// TIA Portal V19 export
FUNCTION_BLOCK "DrvSafeSinaSTlg30"   // FB5, F_LAD
TITLE = SINAMICS S Safety Integrated Functions
// The library includes fail-safe S7 blocks to implement various applications in conjunction with S7-1200F, S7-1500F, S7-1500F Software Controller, SINUMERIK ONE and SINAMICS or SIMATIC Micro Drive coupled via PROFIsafe.
// Additional information in the application example "SIMATIC - Failsafe library LDrvSafe to control the Safety Integrated functions of the SINAMICS drive family"
// stored: IsIECCheckEnabled true, Namespace Safety
   VAR_INPUT
      ack { ExternalAccessible := 'False'; ExternalVisible := 'False'; ExternalWritable := 'False'} : Bool := false;   // Acknowledge bit
      sto { ExternalAccessible := 'False'; ExternalVisible := 'False'; ExternalWritable := 'False'} : Bool := true;   // 1: Deselect STO 0: Select STO
      ss1 { ExternalAccessible := 'False'; ExternalVisible := 'False'; ExternalWritable := 'False'} : Bool := true;   // 1: Deselect SS1 0: Select SS1
      sls { ExternalAccessible := 'False'; ExternalVisible := 'False'; ExternalWritable := 'False'} : Bool := true;   // 1: Deselect SLS 0: Select SLS
      statusWord { ExternalAccessible := 'False'; ExternalVisible := 'False'; ExternalWritable := 'False'} : "Safety.LDrvSafe_typeSinaSTlg30Status";   // PROFIsafe status telegram of the drive
   END_VAR
   VAR_OUTPUT
      status { ExternalAccessible := 'False'; ExternalVisible := 'False'; ExternalWritable := 'False'} : "Safety.typeSafetyDrive";
      controlWord { ExternalAccessible := 'False'; ExternalVisible := 'False'; ExternalWritable := 'False'} : "Safety.LDrvSafe_typeSinaSTlg30Control";   // PROFIsafe control telegram of the drive
   END_VAR
   VAR
      instLDrvSafeSinaSTlg30Status { ExternalAccessible := 'False'; ExternalVisible := 'False'; ExternalWritable := 'False'} : "Safety.LDrvSafe_SinaSTlg30Status";   // Instance data for status telegram
      instLDrvSafeSinaSTlg30Control { ExternalAccessible := 'False'; ExternalVisible := 'False'; ExternalWritable := 'False'} : "Safety.LDrvSafe_SinaSTlg30Control";   // Instance data for control telegram
   END_VAR
BEGIN

REGION Network 1: Control telegram
   // This block controls the safety integrated functions of a SINAMICS S drive via PROFIsafe telegram 30
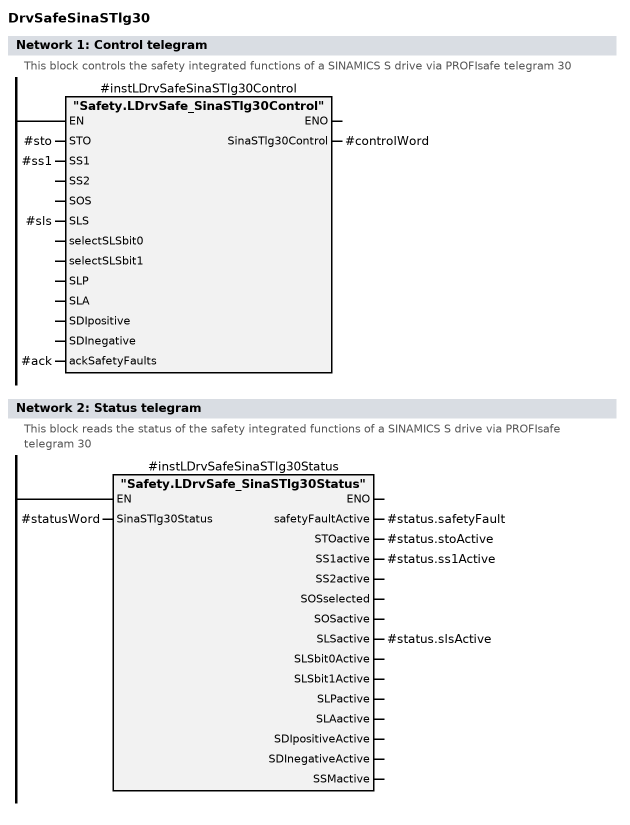
   RUNG wire#powerrail
      #instLDrvSafeSinaSTlg30Control(STO := #sto, SS1 := #ss1, SS2 :=, SOS :=, SLS := #sls, selectSLSbit0 :=, selectSLSbit1 :=, SLP :=, SLA :=, SDIpositive :=, SDInegative :=, ackSafetyFaults := #ack, SinaSTlg30Control => #controlWord)
   END_RUNG
   // the same network as SCL:
   #instLDrvSafeSinaSTlg30Control(STO := #sto,   // "Safety.LDrvSafe_SinaSTlg30Control"
                           SS1 := #ss1,
                           SLS := #sls,
                           ackSafetyFaults := #ack,
                           SinaSTlg30Control => #controlWord);
END_REGION

REGION Network 2: Status telegram
   // This block reads the status of the safety integrated functions of a SINAMICS S drive via PROFIsafe telegram 30
   RUNG wire#powerrail
      #instLDrvSafeSinaSTlg30Status(SinaSTlg30Status := #statusWord, safetyFaultActive => #status.safetyFault, STOactive => #status.stoActive, SS1active => #status.ss1Active, SS2active =>, SOSselected =>, SOSactive =>, SLSactive => #status.slsActive, SLSbit0Active =>, SLSbit1Active =>, SLPactive =>, SLAactive =>, SDIpositiveActive =>, SDInegativeActive =>, SSMactive =>)
   END_RUNG
   // the same network as SCL:
   #instLDrvSafeSinaSTlg30Status(SinaSTlg30Status := #statusWord,   // "Safety.LDrvSafe_SinaSTlg30Status"
                           safetyFaultActive => #status.safetyFault,
                           STOactive => #status.stoActive,
                           SS1active => #status.ss1Active,
                           SLSactive => #status.slsActive);
END_REGION
END_FUNCTION_BLOCK
